(* CODESYS project FB_TESTING.action_test.xml

Project tree, tasks and I/O mapping:
*)

// action_test
ACTION action_test:
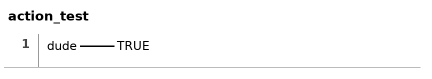
// NETWORK 1
TRUE := dude;
END_ACTION
